{attribute 'qualified_only'}
VAR_GLOBAL
	EL1088_IN	AT%I*	:BYTE;
	EL2088_OUT	AT%Q*	:BYTE;
END_VAR

(* stored: Version 1.1.0.1, ProductVersion 3.1.4024.12
   GVL GVL: Id {5c0516a1-dc14-4f57-bb87-ec442e63ea89} *)
